(* IEC 61131-3 sources: POMIRTS_lab3/AS/Library/MTFlow/V1.00.3, 2 files *)

(* ---- MTFlow.typ ---- *)
(********************************************************************
 * COPYRIGHT -- Bernecker + Rainer
 ********************************************************************
 * Library: MTFlow
 * File: MTFlow.typ
 * Author: B&R
 ********************************************************************
 * Data types of library MTFlow
 ********************************************************************)

TYPE
	MTFlowStatusEnum :
		( (*Status information*)
		mtERR_ORIFICE_TYPE_NOT_VALID := 36740, (*Error: Definition of orifice type invalid*)
		mtERR_NOZZLE_TYPE_NOT_VALID := 36741, (*Error: Definition of nozzle type invalid*)
		mtERR_VENTURI_TYPE_NOT_VALID := 36742, (*Error: Definition of venturi pipe type invalid*)
		mtERR_NEWTON_ITERATION_FAILED := 36743, (*Error: Iteration process failed to produce a valid solution*)
		mtERR_PRESSURE_RATIO_NOT_VALID := 36744, (*Error: Pressure ratio is outside valid range*)
		mtWARN_BORE_DIAMETER_NOT_VALID := 36730, (*Warning: Diameter of throttle unit outside valid range*)
		mtWARN_PIPE_DIAMETER_NOT_VALID := 36731, (*Warning: Pipe diameter outside valid range*)
		mtWARN_DIAMETER_RATIO_NOT_VALID := 36732, (*Warning: Diameter ratio outside valid range*)
		mtWARN_REYNOLDS_OUT_VALID_RANGE := 36733, (*Warning: Reynolds number is outside the valid range*)
		mtWARN_NEWTON_MAX_IT_REACHED := 36734 (*Warning: The maximum number of iterations has been reached*)
		);
	MTFlowOrificeEnum :
		( (*Orifice type*)
		mtORIFICE_CORNER_TAPPING := 1, (*Orifice plate with corner pressure tappings*)
		mtORIFICE_D_D05_TAPPING := 2, (*Orifice plate with D and D/2 pressure tappings*)
		mtORIFICE_FLANGE_TAPPING := 3 (*Orifice plate with flange pressure tappings*)
		);
	MTFlowNozzleEnum :
		( (*Nozzle type*)
		mtNOZZLE_ISA_1932 := 1, (*ISA 1932 nozzle*)
		mtNOZZLE_LONG_RADIUS := 2, (*Long radius nozzle*)
		mtNOZZLE_VENTURI := 3 (*Venturi nozzle*)
		);
	MTFlowVenturiEnum :
		( (*Venturi tube type*)
		mtVENTURI_CAST := 1, (*Classical Venturi tube with an "as cast" convergent section*)
		mtVENTURI_MACHINED := 2, (*Classical Venturi tube with a machined convergent section*)
		mtVENTURI_ROUGH_WELDED := 3, (*Classical Venturi tube with a rough-welded sheet-iron convergent section*)
		mtVENTURI_USER_SPECIFIC := 4 (*User specific venturi tube, Discharge coefficient has to be defined (no limitations) *)
		);
	MTFlowInternalType : 	STRUCT
		Iterations : UINT := 0; (*Data for internal use.*)
		ItSuccess : BOOL := 0; (*Data for internal use.*)
		ItStartValue : LREAL; (*Data for internal use.*)
		ItStepControl : LREAL := 1.0; (*Data for internal use.*)
		NewtonEps : LREAL; (*Data for internal use.*)
		MaxIt : UINT := 200; (*Data for internal use.*)
		CycleTime : REAL; (*Task cycle time. Unit: [s].*)
		Bootkey : UDINT := 0; (*Data for internal use.*)
	END_STRUCT;
END_TYPE

(* ---- MTFlow.fun ---- *)
(********************************************************************
 * COPYRIGHT -- Bernecker + Rainer
 ********************************************************************
 * Library: MTFlow
 * File: MTFlow.fun
 * Author: B&R
 ********************************************************************
 * Functions and function blocks of library MTFlow
 ********************************************************************)

 FUNCTION_BLOCK MTFlowOrifice (*Function block to measure mass flow with orifices according to EN ISO 5167-2*)
	VAR_INPUT
		Enable : BOOL; (*Enable / disable function block*)
		OrificeType : MTFlowOrificeEnum; (*Kind of pressure tapping (defined with Quotients of distance (up-/downstream)*)
		DiameterPipe : LREAL; (*Pipe diameter in mm*)
		DiameterBore : LREAL; (*Bore diameter in mm*)
		DensityUpstream : LREAL; (*Density upstream in kg/mł*)
		KinViscUpstream : LREAL; (*Kinematic viscosity upstream in m˛/s*)
		EnableCompressibility : BOOL; (*Enable / disable consider compressibility of fluid*)
		IsentropicExponent : LREAL; (*Isentropic exponent*)
		PressureUpstream : LREAL; (*Upstream pressure in bar*)
		PressureDownstream : LREAL; (*Downstream pressure in bar*)
	END_VAR
	VAR_OUTPUT
		Active : BOOL; (*Function block active*)
		Error : BOOL; (*Function block error *)
		StatusID : MTFlowStatusEnum; (*Status ID*)
		DiameterRatio : LREAL; (*Diameter ratio DiameterBore/DiameterPipe*)
		ExpansionFactor : LREAL; (*Expansion factor*)
		ReynoldsDiameterPipe : LREAL; (*Reynolds number with respect to pipe diameter*)
		DischargeCoefficient : LREAL; (*Discharge coefficient, Reader-Harris/Gallager equation*)
		FlowVelocityPipe : LREAL; (*Mean axial velocity of the fluid in the pipe in m/s*)
		VolumeFlow : LREAL; (*Volume flow rate in mł/s*)
		MassFlow : LREAL; (*Mass flow rate in kg/s*)
		DistanceQuotientUpstream : LREAL; (*Quotient of the distance of the upstream tapping from the upstream face of the plate and the pipe diameter*)
		DistanceQuotientDownstream : LREAL; (*Quotient of the distance of the downstream tapping from the downstream face of the plate and the pipe diameter (downstream spacing from the downstream face)*)
	END_VAR
	VAR
		Internal : MTFlowInternalType; (*Internal parameter*)
	END_VAR
END_FUNCTION_BLOCK

 FUNCTION_BLOCK MTFlowNozzle (*Function block to measure mass flow with nozzles according to EN ISO 5167-3*)
	VAR_INPUT
		Enable : BOOL; (*Enable / disable function block*)
		NozzleType : MTFlowNozzleEnum; (*Define nozzle type*)
		DiameterPipe : LREAL; (*Pipe diameter in mm*)
		DiameterBore : LREAL; (*Bore diameter in mm*)
		DensityUpstream : LREAL; (*Density upstream in kg/mł*)
		KinViscUpstream : LREAL; (*Kinematic viscosity upstream in m˛/s*)
		EnableCompressibility : BOOL; (*Enable / disable consider compressibility of fluid*)
		IsentropicExponent : LREAL; (*Isentropic exponent*)
		PressureUpstream : LREAL; (*Upstream pressure in bar*)
		PressureDownstream : LREAL; (*Downstream pressure in bar*)
	END_VAR
	VAR_OUTPUT
		Active : BOOL; (*Function block active*)
		Error : BOOL; (*Function block error *)
		StatusID : MTFlowStatusEnum; (*Status ID*)
		DiameterRatio : LREAL; (*Diameter ratio DiameterBore/DiameterPipe*)
		ExpansionFactor : LREAL; (*Expansion factor*)
		ReynoldsDiameterPipe : LREAL; (*Reynolds number with respect to pipe diameter*)
		DischargeCoefficient : LREAL; (*Discharge coefficient, Reader-Harris/Gallager equation*)
		FlowVelocityPipe : LREAL; (*Mean axial velocity of the fluid in the pipe in m/s*)
		VolumeFlow : LREAL; (*Volume flow rate in mł/s*)
		MassFlow : LREAL; (*Mass flow rate in kg/s*)
	END_VAR
	VAR
		Internal : MTFlowInternalType; (*Internal parameter*)
	END_VAR
END_FUNCTION_BLOCK

 FUNCTION_BLOCK MTFlowVenturi (*Function block to measure mass flow with venturi tubes according to EN ISO 5167-4 *)
	VAR_INPUT
		Enable : BOOL; (*Enable / disable function block*)
		VenturiType : MTFlowVenturiEnum; (*Define type of venturi tube*)
		DiameterPipe : LREAL; (*Pipe diameter in mm*)
		DiameterBore : LREAL; (*Bore diameter in mm*)
		DensityUpstream : LREAL; (*Density upstream in kg/mł*)
		KinViscUpstream : LREAL; (*Kinematic viscosity upstream in m˛/s*)
		EnableCompressibility : BOOL; (*Enable / disable consider compressibility of fluid*)
		IsentropicExponent : LREAL; (*Isentropic exponent*)
		PressureUpstream : LREAL; (*Upstream pressure in bar*)
		PressureDownstream : LREAL; (*Downstream pressure in bar*)
		DischargeCoefficientExternal : LREAL; (*External DischargeCoefficient if VenturiType == mtVENTURI_USER_SPECIFIC*)
	END_VAR
	VAR_OUTPUT
		Active : BOOL; (*Function block active*)
		Error : BOOL; (*Function block error *)
		StatusID : MTFlowStatusEnum; (*Status ID*)
		DiameterRatio : LREAL; (*Diameter ratio DiameterBore/DiameterPipe*)
		ExpansionFactor : LREAL; (*Expansion factor*)
		ReynoldsDiameterPipe : LREAL; (*Reynolds number with respect to pipe diameter*)
		DischargeCoefficient : LREAL; (*Discharge coefficient, Reader-Harris/Gallager equation*)
		FlowVelocityPipe : LREAL; (*Mean axial velocity of the fluid in the pipe in m/s*)
		VolumeFlow : LREAL; (*Volume flow rate in mł/s*)
		MassFlow : LREAL; (*Mass flow rate in kg/s*)
	END_VAR
END_FUNCTION_BLOCK
